Fanuc KAREL source: CNV_CONF_STR.kl

PROGRAM T
%NOLOCKGROUP
VAR
 v0 : CONFIG
 v1 : STRING[40]
BEGIN
 CNV_CONF_STR(v0, v1)
END T
